FUNCTION_BLOCK CRANE2_DECIDER (* Service Interface Function Block Type *)
  (* Standard: 61499-2 *)
  (* Version 1.0, 2019-03-16, adeel *)
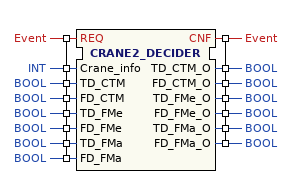
  EVENT_INPUT
    REQ WITH Crane_info, TD_CTM, FD_CTM, TD_FMe, FD_FMe, TD_FMa, FD_FMa; (* Service Request *)
  END_EVENT
  EVENT_OUTPUT
    CNF WITH TD_CTM_O, FD_CTM_O, TD_FMe_O, FD_FMe_O, TD_FMa_O, FD_FMa_O; (* Confirmation of Requested Service *)
  END_EVENT
  VAR_INPUT
    Crane_info : INT;
    TD_CTM : BOOL;
    FD_CTM : BOOL;
    TD_FMe : BOOL;
    FD_FMe : BOOL;
    TD_FMa : BOOL;
    FD_FMa : BOOL;
  END_VAR
  VAR_OUTPUT
    TD_CTM_O : BOOL;
    FD_CTM_O : BOOL;
    TD_FMe_O : BOOL;
    FD_FMe_O : BOOL;
    TD_FMa_O : BOOL;
    FD_FMa_O : BOOL;
  END_VAR
  SERVICE APPLICATION/RESOURCE (* Service Interface Function Block Type *)
    SEQUENCE normal_establishment
      APPLICATION.INIT+(PARAMS) -> RESOURCE.initialize(PARAMS) -> APPLICATION.INITO+();
    END_SEQUENCE
    SEQUENCE unsuccessful_establishment
      APPLICATION.INIT+(PARAMS) -> RESOURCE.initialize(PARAMS) -> APPLICATION.INITO-(STATUS);
    END_SEQUENCE
    SEQUENCE request_confirm
      APPLICATION.REQ+(SD) -> RESOURCE.request(SD) -> APPLICATION.CNF+(RD);
    END_SEQUENCE
    SEQUENCE request_inhibited
      APPLICATION.REQ-(SD) -> APPLICATION.CNF-(STATUS);
    END_SEQUENCE
    SEQUENCE request_error
      APPLICATION.REQ+(SD) -> RESOURCE.request(SD) -> APPLICATION.CNF-(STATUS);
    END_SEQUENCE
    SEQUENCE indication_response
      RESOURCE.indicate(RD) -> APPLICATION.IND+(RD);
      APPLICATION.RSP(QI,SD) -> RESOURCE.response(QI,SD);
    END_SEQUENCE
    SEQUENCE indication_inhibited
      RESOURCE.indicate(RD,QI=FALSE) -> RESOURCE.inhibited();
    END_SEQUENCE
    SEQUENCE error_indication
      RESOURCE.error(STATUS) -> APPLICATION.IND-(STATUS);
    END_SEQUENCE
    SEQUENCE application_initiated_termination
      APPLICATION.INIT-() -> RESOURCE.terminate() -> APPLICATION.INITO-(STATUS);
    END_SEQUENCE
    SEQUENCE resource_initiated_termination
      -> APPLICATION.INITO-(STATUS);
    END_SEQUENCE
  END_SERVICE
END_FUNCTION_BLOCK
